// TIA Portal V20 export
TYPE "LER_typeAlignThetaCalibrationInterface"
// stored: Access Published
   STRUCT
      commands : "LER_typeAlignThetaCalibrationCommands";
      monitoring : "LER_typeAlignThetaCalibrationMonitoring";
      configuration : "LER_typeAlignThetaCalibrationConfiguration";
   END_STRUCT;
END_TYPE
